FUNCTION_BLOCK FB_GaugeSelection EXTENDS FB_GaugeBase
VAR_INPUT
    st_defaultGauge : ST_VG;
    st_secondGauge : ST_VG;
END_VAR
VAR_OUTPUT
    IG : ST_VG;
END_VAR
VAR
END_VAR

IF NOT st_defaultGauge.xPRESS_OK AND st_secondGauge.xPRESS_OK THEN
    IG := st_secondGauge;
ELSE
    IG := st_defaultGauge;
END_IF

END_FUNCTION_BLOCK

(* stored: Version 1.1.0.1
   POU FB_GaugeSelection: Id {d0430b83-40b0-475f-aa09-4e109be9ff76}, SpecialFunc None *)
